(* PLC project Plc Structured Text Cheatsheet, CODESYS CODESYS V3.5 SP16, author Toni Kucic *)
(* stored: creationDateTime 2022-05-27T13:55:14.4433933, version 1.0, modificationDateTime 2022-05-27T13:55:00.8059953, organization TK Automation *)
(* Cheatsheet for programming a PLC in IEC61131-3 Structured text. Contains usage of operators and common functions. *)

TYPE dtTestStruct : STRUCT
  dummy1 : USINT := 255;
  Elem1 : INT := -1;
  Id : DWORD := 215215126;
  IdText : STRING := 'Testing for speed';
  dummy2 : ARRAY[0..11] OF DWORD;
  dummy4 : BOOL := FALSE;
  dummy5 : STRING(255) := 'Big array';
  dummy6 : LINT := 1211212723838939;
END_STRUCT;
END_TYPE

PROGRAM floatingPointOperations
  VAR CONSTANT
    cNrRuns : USINT := 5;
    cRepeatCalcTimes : UDINT := 10000000;  (* 10 Million times *)
  END_VAR
  VAR
    vResultsA : ARRAY[0..cNrRuns] OF LTIME;  (* Boiler plate variables for test *)
    vResultsB : ARRAY[0..cNrRuns] OF LTIME;
    vResultsC : ARRAY[0..cNrRuns] OF LTIME;
    vResultsD : ARRAY[0..cNrRuns] OF LTIME;
    vResultsE : ARRAY[0..cNrRuns] OF LTIME;
    vResultsF : ARRAY[0..cNrRuns] OF LTIME;
    vResultsG : ARRAY[0..cNrRuns] OF LTIME;
    vResultsH : ARRAY[0..cNrRuns] OF LTIME;
    vResultsI : ARRAY[0..cNrRuns] OF LTIME;
    vResultsAAVG : LTIME;
    vResultsBAVG : LTIME;
    vResultsCAVG : LTIME;
    vResultsDAVG : LTIME;
    vResultsEAVG : LTIME;
    vResultsFAVG : LTIME;
    vResultsGAVG : LTIME;
    vResultsHAVG : LTIME;
    vResultsIAVG : LTIME;
    vWayAOldTime : LTIME;
    vWayBOldTime : LTIME;
    vWayCOldTime : LTIME;
    vWayDOldTime : LTIME;
    vWayEOldTime : LTIME;
    vWayFOldTime : LTIME;
    vWayGOldTime : LTIME;
    vWayHOldTime : LTIME;
    vWayIOldTime : LTIME;
    vWayAExecTime : LTIME;
    vWayBExecTime : LTIME;
    vWayCExecTime : LTIME;
    vWayDExecTime : LTIME;
    vWayEExecTime : LTIME;
    vWayFExecTime : LTIME;
    vWayGExecTime : LTIME;
    vWayHExecTime : LTIME;
    vWayIExecTime : LTIME;
    i : UDINT;
    vRunsCompleted : USINT := 0;
    vInteger1 : INT := 1234;  (* Test vars *)
    vInteger2 : INT := 4231;
    vReal1 : REAL := 1234.4231;
    vReal2 : REAL := 4231.1234;
    vInteger3 : DINT := 1234;
    vInteger4 : DINT := 4231;
    vResult1 : INT;
    vResult2 : REAL;
    vResult3 : DINT;
    vResult4 : INT;
    vResult5 : REAL;
    vResult6 : DINT;
    vResult7 : INT;
    vResult8 : REAL;
    vResult9 : DINT;
  END_VAR

            IF vRunsCompleted > cNrRuns THEN
	vResultsAAVG := calcAvg(vResultsA); //Time to add two integers 10 milion times
	vResultsBAVG := calcAvg(vResultsB); //Time to add two reals 10 milion times
	vResultsCAVG := calcAvg(vResultsC); //Time to add two DINTs (32b INT) 10 milion times
	vResultsDAVG := calcAvg(vResultsD); //Time to multiply two integers 10 milion times
	vResultsEAVG := calcAvg(vResultsE); //Time to multiply two reals 10 milion times
	vResultsFAVG := calcAvg(vResultsF); //Time to multiply two DINTs (32b INT) 10 milion times
	vResultsGAVG := calcAvg(vResultsG); //Time to divide two integers 10 milion times
	vResultsHAVG := calcAvg(vResultsH); //Time to divide two reals 10 milion times
	vResultsIAVG := calcAvg(vResultsI); //Time to divide two DINTs (32b INT) 10 milion times
	RETURN;
END_IF

//------------CALCULATION A -------------------
vWayAOldTime := LTIME();
FOR i:= 0 TO cRepeatCalcTimes DO
	vResult1 := vInteger1 + vInteger2;
END_FOR
vWayAExecTime := LTIME() - vWayAOldTime;

//------------CALCULATION B -------------------
vWayBOldTime := LTIME();
FOR i:= 0 TO cRepeatCalcTimes DO
	vResult2 := vReal1 + vReal2;
END_FOR
vWayBExecTime := LTIME() - vWayBOldTime;

//------------CALCULATION C -------------------
vWayCOldTime := LTIME();
FOR i:= 0 TO cRepeatCalcTimes DO
	vResult3 := vInteger3 + vInteger4;
END_FOR
vWayCExecTime := LTIME() - vWayCOldTime;

//------------CALCULATION D -------------------
vWayDOldTime := LTIME();
FOR i:= 0 TO cRepeatCalcTimes DO
	vResult4 := vInteger1 * vInteger2;
END_FOR
vWayDExecTime := LTIME() - vWayDOldTime;

//------------CALCULATION E -------------------
vWayEOldTime := LTIME();
FOR i:= 0 TO cRepeatCalcTimes DO
	vResult5 := vReal1 * vReal2;
END_FOR
vWayEExecTime := LTIME() - vWayEOldTime;

//------------CALCULATION F -------------------
vWayFOldTime := LTIME();
FOR i:= 0 TO cRepeatCalcTimes DO
	vResult6 := vInteger3 * vInteger4;
END_FOR
vWayFExecTime := LTIME() - vWayFOldTime;

//------------CALCULATION G -------------------
vWayGOldTime := LTIME();
FOR i:= 0 TO cRepeatCalcTimes DO
	vResult7 := vInteger1 / vInteger2;
END_FOR
vWayGExecTime := LTIME() - vWayGOldTime;

//------------CALCULATION H -------------------
vWayHOldTime := LTIME();
FOR i:= 0 TO cRepeatCalcTimes DO
	vResult8 := vReal1 / vReal2;
END_FOR
vWayHExecTime := LTIME() - vWayHOldTime;

//------------CALCULATION I -------------------
vWayIOldTime := LTIME();
FOR i:= 0 TO cRepeatCalcTimes DO
	vResult9 := vInteger3 / vInteger4;
END_FOR
vWayIExecTime := LTIME() - vWayIOldTime;


//------------CATCH RESULTS---------------------
vResultsA[vRunsCompleted] := vWayAExecTime;
vResultsB[vRunsCompleted] := vWayBExecTime;
vResultsC[vRunsCompleted] := vWayCExecTime;
vResultsD[vRunsCompleted] := vWayDExecTime;
vResultsE[vRunsCompleted] := vWayEExecTime;
vResultsF[vRunsCompleted] := vWayFExecTime;
vResultsG[vRunsCompleted] := vWayGExecTime;
vResultsH[vRunsCompleted] := vWayHExecTime;
vResultsI[vRunsCompleted] := vWayIExecTime;
vRunsCompleted := vRunsCompleted + 1;

          
END_PROGRAM

FUNCTION addTwoInts : INT
  VAR_IN_OUT
    int1 : INT;
    int2 : INT;
  END_VAR

            addTwoInts := int1 + int2;
          
END_FUNCTION

PROGRAM FunctionOverhead
  VAR CONSTANT
    cNrRuns : USINT := 4;
    cRepeatCalcTimes : UDINT := 10000000;  (* Million times *)
  END_VAR
  VAR
    vResultsA : ARRAY[0..cNrRuns] OF LTIME;  (* Boiler plate variables for test *)
    vResultsB : ARRAY[0..cNrRuns] OF LTIME;
    vResultsC : ARRAY[0..cNrRuns] OF LTIME;
    vResultsAAVG : LTIME;
    vResultsBAVG : LTIME;
    vResultsCAVG : LTIME;
    vWayAOldTime : LTIME;
    vWayBOldTime : LTIME;
    vWayCOldTime : LTIME;
    vWayAExecTime : LTIME;
    vWayBExecTime : LTIME;
    vWayCExecTime : LTIME;
    i : UDINT;
    vRunsCompleted : USINT := 0;
    vInt1 : INT := 1;  (* Test vars *)
    vInt2 : INT := 2;
    vResult1 : INT;
    vResult2 : INT;
    vResult3 : INT;
  END_VAR

            IF vRunsCompleted > cNrRuns THEN
	vResultsAAVG := calcAvg(vResultsA); //Operands
	vResultsBAVG := calcAvg(vResultsB); //User function
	vResultsCAVG := calcAvg(vResultsC); //PRG method
	RETURN;
END_IF
	
//------------CALCULATION A -------------------
vWayAOldTime := LTIME();
FOR i:= 0 TO cRepeatCalcTimes DO
	vResult1 := vInt1 + vInt2;
END_FOR
vWayAExecTime := LTIME() - vWayAOldTime;

//------------CALCULATION B -------------------
vWayBOldTime := LTIME();
FOR i:= 0 TO cRepeatCalcTimes DO
	vResult2 := addTwoInts(vInt1, vInt2);
END_FOR
vWayBExecTime := LTIME() - vWayBOldTime;

//------------CALCULATION C -------------------
vWayCOldTime := LTIME();
FOR i:= 0 TO cRepeatCalcTimes DO
	vResult3 := addTwoNumbers(vInt1, vInt2);
END_FOR
vWayCExecTime := LTIME() - vWayCOldTime;

//------------CATCH RESULTS---------------------
vResultsA[vRunsCompleted] := vWayAExecTime;
vResultsB[vRunsCompleted] := vWayBExecTime;
vResultsC[vRunsCompleted] := vWayCExecTime;
vRunsCompleted := vRunsCompleted + 1;

          

METHOD addTwoNumbers : INT
  VAR_INPUT
    int1 : INT;
    int2 : INT;
  END_VAR
                  addTwoNumbers := int1 + int2;
                
END_METHOD
END_PROGRAM

PROGRAM ImpactOfDynamicArrays
  VAR CONSTANT
    cNrRuns : USINT := 4;
    cRepeatCalcTimes : UDINT := 1000000;  (* Million times *)
  END_VAR
  VAR
    vResultsA : ARRAY[0..cNrRuns] OF LTIME;  (* Boiler plate variables for test *)
    vResultsB : ARRAY[0..cNrRuns] OF LTIME;
    vResultsAAVG : LTIME;
    vResultsBAVG : LTIME;
    vWayAOldTime : LTIME;
    vWayAExecTime : LTIME;
    vWayBOldTime : LTIME;
    vWayBExecTime : LTIME;
    i : UDINT;
    vRunsCompleted : USINT := 0;
    vAvgTimeFun : LTIME;  (* Test vars *)
    vAvgTimeHardCoded : LTIME;
    vTimes : ARRAY[0..9] OF LTIME := [LTIME#1ms0us0ns, LTIME#2ms0us0ns, LTIME#3ms0us0ns, LTIME#4ms0us0ns, LTIME#5ms0us0ns, LTIME#6ms0us0ns, LTIME#7ms0us0ns, LTIME#8ms0us0ns, LTIME#9ms0us0ns, LTIME#10ms0us0ns];
    j : USINT;
  END_VAR

            IF vRunsCompleted > cNrRuns THEN
	vResultsAAVG := calcAvg(vResultsA);
	vResultsBAVG := calcAvg(vResultsB);
	RETURN;
END_IF
	
//------------CALCULATION A -------------------
vWayAOldTime := LTIME();
FOR i:= 0 TO cRepeatCalcTimes DO
	vAvgTimeFun := calcAvg(vTimes);
END_FOR
vWayAExecTime := LTIME() - vWayAOldTime;

//------------CALCULATION B -------------------
vWayBOldTime := LTIME();
FOR i:= 0 TO cRepeatCalcTimes DO
	vAvgTimeHardCoded := LTIME#0MS;
	FOR j:= 0 TO 9 DO
		vAvgTimeHardCoded := vAvgTimeHardCoded + vTimes[j];
	END_FOR
	vAvgTimeHardCoded := vAvgTimeHardCoded / j;
END_FOR
vWayBExecTime := LTIME() - vWayBOldTime;

//------------CATCH RESULTS---------------------
vResultsA[vRunsCompleted] := vWayAExecTime;
vResultsB[vRunsCompleted] := vWayBExecTime;
vRunsCompleted := vRunsCompleted + 1;

          
END_PROGRAM

PROGRAM ShlVsMemCpy
  VAR CONSTANT
    cNrRuns : USINT := 4;
    cRepeatCalcTimes : UDINT := 1000000;  (* Million times *)
  END_VAR
  VAR
    vResultsA : ARRAY[0..cNrRuns] OF LTIME;  (* Boiler plate variables for test *)
    vResultsB : ARRAY[0..cNrRuns] OF LTIME;
    vResultsAAVG : LTIME;
    vResultsBAVG : LTIME;
    vWayAOldTime : LTIME;
    vWayAExecTime : LTIME;
    vWayBOldTime : LTIME;
    vWayBExecTime : LTIME;
    i : UDINT;
    vRunsCompleted : USINT := 0;
    vSHRInteger : UINT;  (* Test vars *)
    vMcpyInteger : UINT;
    vBuffer : ARRAY[0..1] OF USINT := [16#55, 16#AA];
    vSHLOldTime : LTIME;
    vMcpyOldTime : LTIME;
    vSHLExecTime : LTIME;
    vMcpyExecTime : LTIME;
  END_VAR

            IF vRunsCompleted > cNrRuns THEN
	vResultsAAVG := calcAvg(vResultsA);
	vResultsBAVG := calcAvg(vResultsB);
	RETURN;
END_IF
	

vWayAOldTime := LTIME();
FOR i:= 0 TO cRepeatCalcTimes DO
	//Assemble an UINT from two USINTs using SHR operator
	vSHRInteger := vBuffer[0] + SHL(vBuffer[1],8);
END_FOR
vWayAExecTime := LTIME() - vWayAOldTime;

vWayBOldTime := LTIME();
FOR i:= 0 TO cRepeatCalcTimes DO
	//Assemble an UINT from two USINTs using MemCpy
	MEMUtils.MemCpy(pbyDest:= ADR(vMcpyInteger), pbySrc:= ADR(vBuffer) , dwSize:= SIZEOF(vMcpyInteger));
END_FOR
vWayBExecTime := LTIME() - vWayBOldTime;

//Results
vResultsA[vRunsCompleted] := vWayAExecTime;
vResultsB[vRunsCompleted] := vWayBExecTime;
vRunsCompleted := vRunsCompleted + 1;

          
END_PROGRAM

FUNCTION calcAVG : LTIME
  VAR_INPUT
    {attribute 'variable_length_array' := 'ARRAY[*] OF LTIME'}
    {attribute 'Dimensions' := '1'}
    Results : POINTER TO LTIME;
  END_VAR
  VAR
    i : DINT;
  END_VAR

            FOR i:= LOWER_BOUND(Results,1) TO UPPER_BOUND(Results,1) DO
	calcAvg := calcAvg + Results[i];
END_FOR
calcAvg := calcAvg / i;
RETURN;
          
END_FUNCTION

PROGRAM MemSetVsDataZeero
  VAR CONSTANT
    cNrRuns : USINT := 4;
    cRepeatCalcTimes : UDINT := 1000000;  (* Million times *)
    cEmptyStruct : dtTestStruct;
  END_VAR
  VAR
    vResultsA : ARRAY[0..cNrRuns] OF LTIME;  (* Boiler plate variables for test *)
    vResultsB : ARRAY[0..cNrRuns] OF LTIME;
    vResultsAAVG : LTIME;
    vResultsBAVG : LTIME;
    vWayAOldTime : LTIME;
    vWayAExecTime : LTIME;
    vWayBOldTime : LTIME;
    vWayBExecTime : LTIME;
    i : UDINT;
    vRunsCompleted : USINT := 0;
    vResultStruct1 : dtTestStruct;  (* Test variables *)
    vResultStruct2 : dtTestStruct;
  END_VAR

            IF vRunsCompleted > cNrRuns THEN
	vResultsAAVG := calcAvg(vResultsA);
	vResultsBAVG := calcAvg(vResultsB);
	RETURN;
END_IF
	
//------------CALCULATION A -------------------
vWayAOldTime := LTIME();
FOR i:= 0 TO cRepeatCalcTimes DO
	//RESET STRUCT WITH A EMPTY STRUCT
	vResultStruct1 := cEmptyStruct;
END_FOR
vWayAExecTime := LTIME() - vWayAOldTime;

//------------CALCULATION B -------------------
vWayBOldTime := LTIME();
FOR i:= 0 TO cRepeatCalcTimes DO
	//RESET STRUCT WITH MEM SET
	MEMUtils.MemSet(pbyBuffer:= ADR(vResultStruct2), byValue:= 16#0 , dwSize:= SIZEOF(vResultStruct2));
END_FOR
vWayBExecTime := LTIME() - vWayBOldTime;

//------------CATCH RESULTS---------------------
vResultsA[vRunsCompleted] := vWayAExecTime;
vResultsB[vRunsCompleted] := vWayBExecTime;
vRunsCompleted := vRunsCompleted + 1;

          
END_PROGRAM

PROGRAM execSpeedOfLanguageTypes
  VAR CONSTANT
    cNrRuns : USINT := 4;
    cRepeatCalcTimes : UDINT := 10000000;  (* Million times *)
  END_VAR
  VAR
    vResultsA : ARRAY[0..cNrRuns] OF LTIME;  (* Boiler plate variables for test *)
    vResultsB : ARRAY[0..cNrRuns] OF LTIME;
    vResultsC : ARRAY[0..cNrRuns] OF LTIME;
    vResultsAAVG : LTIME;
    vResultsBAVG : LTIME;
    vResultsCAVG : LTIME;
    vWayAOldTime : LTIME;
    vWayBOldTime : LTIME;
    vWayCOldTime : LTIME;
    vWayAExecTime : LTIME;
    vWayBExecTime : LTIME;
    vWayCExecTime : LTIME;
    i : UDINT;
    vRunsCompleted : USINT := 0;
    vInt1 : INT := 1;  (* Test vars *)
    vInt2 : INT := 2;
    vResult1 : INT;
    vResult2 : INT;
    vResult3 : INT;
  END_VAR

            IF vRunsCompleted > cNrRuns THEN
	vResultsAAVG := calcAvg(vResultsA); //User function Ladder
	vResultsBAVG := calcAvg(vResultsB); //User function ST
	vResultsCAVG := calcAvg(vResultsC); //User function FBD
	RETURN;
END_IF
	
//------------CALCULATION A -------------------
vWayAOldTime := LTIME();
FOR i:= 0 TO cRepeatCalcTimes DO
	vResult1 := addTwoIntsLadder(vInt1, vInt2);
END_FOR
vWayAExecTime := LTIME() - vWayAOldTime;

//------------CALCULATION B -------------------
vWayBOldTime := LTIME();
FOR i:= 0 TO cRepeatCalcTimes DO
	vResult2 := addTwoIntsST(vInt1, vInt2);
END_FOR
vWayBExecTime := LTIME() - vWayBOldTime;

//------------CALCULATION C -------------------
vWayCOldTime := LTIME();
FOR i:= 0 TO cRepeatCalcTimes DO
	vResult3 := addTwoIntsFBD(vInt1, vInt2);
END_FOR
vWayCExecTime := LTIME() - vWayCOldTime;

//------------CATCH RESULTS---------------------
vResultsA[vRunsCompleted] := vWayAExecTime;
vResultsB[vRunsCompleted] := vWayBExecTime;
vResultsC[vRunsCompleted] := vWayCExecTime;
vRunsCompleted := vRunsCompleted + 1;

          
END_PROGRAM

FUNCTION addTwoIntsLadder : INT
  VAR_INPUT
    Int1 : INT;
    Int2 : INT;
  END_VAR

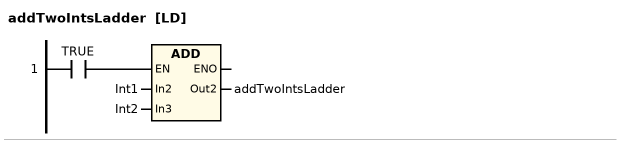
(* LD diagram, written out as Structured Text *)

IF TRUE THEN addTwoIntsLadder := Int1 + Int2; END_IF;
END_FUNCTION

FUNCTION addTwoIntsST : INT
  VAR_INPUT
    int1 : INT;
    int2 : INT;
  END_VAR

            addTwoIntsST := int1 + int2;
          
END_FUNCTION

FUNCTION addTwoIntsFBD : INT
  VAR_INPUT
    int1 : INT;
    int2 : INT;
  END_VAR

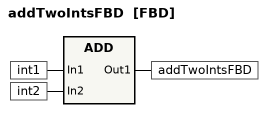
(* FBD diagram, written out as Structured Text *)
addTwoIntsFBD := int1 + int2;
END_FUNCTION

PROGRAM stringOperations
  VAR CONSTANT
    cNrRuns : USINT := 4;
    cRepeatCalcTimes : UDINT := 1000;  (* Million times *)
  END_VAR
  VAR
    vResultsA : ARRAY[0..cNrRuns] OF LTIME;  (* Boiler plate variables for test *)
    vResultsB : ARRAY[0..cNrRuns] OF LTIME;
    vResultsC : ARRAY[0..cNrRuns] OF LTIME;
    vResultsD : ARRAY[0..cNrRuns] OF LTIME;
    vResultsE : ARRAY[0..cNrRuns] OF LTIME;
    vResultsF : ARRAY[0..cNrRuns] OF LTIME;
    vResultsAAVG : LTIME;  (* Time to copy a string[255] 1000 times *)
    vResultsBAVG : LTIME;  (* Time to copy a string 1000 times *)
    vResultsCAVG : LTIME;  (* Time to concatenate 1000 characters with STRING *)
    vResultsDAVG : LTIME;  (* Time to concatenate 1000 characters with STRING[255] *)
    vResultsEAVG : LTIME;  (* Time to copy a BYTE 1000 times *)
    vResultsFAVG : LTIME;  (* Time to copy an array of 255 BYTE 1000 times *)
    vWayAOldTime : LTIME;
    vWayBOldTime : LTIME;
    vWayCOldTime : LTIME;
    vWayDOldTime : LTIME;
    vWayEOldTime : LTIME;
    vWayFOldTime : LTIME;
    vWayAExecTime : LTIME;
    vWayBExecTime : LTIME;
    vWayCExecTime : LTIME;
    vWayDExecTime : LTIME;
    vWayEExecTime : LTIME;
    vWayFExecTime : LTIME;
    i : UDINT;
    vRunsCompleted : USINT := 0;
    vString1 : STRING(255) := 'Test string1';  (* Test vars *)
    vString2 : STRING := 'Test string2';
    vString3 : STRING := 'a';
    vString4 : STRING := 'a';
    vByte : BYTE := 16#FF;
    vArrByte : ARRAY[0..255] OF BYTE;
    vResult1 : STRING(255);
    vResult2 : STRING;
    vResult3 : STRING;
    vResult4 : STRING(255);
    vResult5 : BYTE;
    vResult6 : ARRAY[0..255] OF BYTE;
    vSizes : ARRAY[0..3] OF UDINT;
  END_VAR

            IF vRunsCompleted > cNrRuns THEN
	vResultsAAVG := calcAvg(vResultsA); //Time to copy a string[255] 1000 times
	vResultsBAVG := calcAvg(vResultsB); //Time to copy a string 1000 times
	vResultsCAVG := calcAvg(vResultsC); //Time to concatenate 1000 characters with STRING
	vResultsDAVG := calcAvg(vResultsD); //Time to concatenate 1000  characters with STRING[255]
	vResultsEAVG := calcAvg(vResultsE); //Time to move a byte 1000 times
	vResultsFAVG := calcAvg(vResultsF); //Time to copy an array of 255 BYTE 1000 times
	RETURN;
END_IF

vSizes[0] := SIZEOF(vString1); //Size is 255 characters + zero char
vSizes[1] := SIZEOF(vString2); //Size is 80 characters + zero char, default if no size specified
vSizes[2] := SIZEOF(vResult3); //Size is 81, even though we concatenated 1000 characters. The rest were chopped off
vSizes[3] := SIZEOF(vResult4); //Size is expected 256, other 744 characters chopped off

//------------CALCULATION A -------------------
vWayAOldTime := LTIME();
FOR i:= 0 TO cRepeatCalcTimes DO
	vResult1 := vString1;
END_FOR
vWayAExecTime := LTIME() - vWayAOldTime;

//------------CALCULATION B -------------------
vWayBOldTime := LTIME();
FOR i:= 0 TO cRepeatCalcTimes DO
	vResult2 := vString2;
END_FOR
vWayBExecTime := LTIME() - vWayBOldTime;

//------------CALCULATION C -------------------
vWayCOldTime := LTIME();
FOR i:= 0 TO cRepeatCalcTimes DO
	vResult3 := CONCAT(vResult3, vString3);
END_FOR
vWayCExecTime := LTIME() - vWayCOldTime;

//------------CALCULATION D -------------------
vWayDOldTime := LTIME();
FOR i:= 0 TO cRepeatCalcTimes DO
	vResult4 := CONCAT(vResult4, vString4);
END_FOR
vWayDExecTime := LTIME() - vWayDOldTime;

//------------CALCULATION E -------------------
vWayEOldTime := LTIME();
FOR i:= 0 TO cRepeatCalcTimes DO
	vResult5 := vByte;
END_FOR
vWayEExecTime := LTIME() - vWayEOldTime;

//------------CALCULATION F -------------------
vWayFOldTime := LTIME();
FOR i:= 0 TO cRepeatCalcTimes DO
	vResult6 := vArrByte;
END_FOR
vWayFExecTime := LTIME() - vWayFOldTime;

//------------CATCH RESULTS---------------------
vResultsA[vRunsCompleted] := vWayAExecTime;
vResultsB[vRunsCompleted] := vWayBExecTime;
vResultsC[vRunsCompleted] := vWayCExecTime;
vResultsD[vRunsCompleted] := vWayDExecTime;
vResultsE[vRunsCompleted] := vWayEExecTime;
vResultsF[vRunsCompleted] := vWayFExecTime;
vRunsCompleted := vRunsCompleted + 1;

          
END_PROGRAM

PROGRAM checkingBools
  VAR CONSTANT
    cNrRuns : USINT := 5;
    cRepeatCalcTimes : UDINT := 10000;  (* 10 Million times *)
  END_VAR
  VAR
    vResultsA : ARRAY[0..cNrRuns] OF LTIME;  (* Boiler plate variables for test *)
    vResultsB : ARRAY[0..cNrRuns] OF LTIME;
    vResultsC : ARRAY[0..cNrRuns] OF LTIME;
    vResultsD : ARRAY[0..cNrRuns] OF LTIME;
    vResultsE : ARRAY[0..cNrRuns] OF LTIME;
    vResultsAAVG : LTIME;
    vResultsBAVG : LTIME;
    vResultsCAVG : LTIME;
    vResultsDAVG : LTIME;
    vResultsEAVG : LTIME;
    vWayAOldTime : LTIME;
    vWayBOldTime : LTIME;
    vWayCOldTime : LTIME;
    vWayDOldTime : LTIME;
    vWayEOldTime : LTIME;
    vWayAExecTime : LTIME;
    vWayBExecTime : LTIME;
    vWayCExecTime : LTIME;
    vWayDExecTime : LTIME;
    vWayEExecTime : LTIME;
    i : UDINT;
    vRunsCompleted : USINT := 0;
    vBool : BOOL := TRUE;  (* Test vars *)
    vResult : BOOL;
    vCounter : UINT := 0;
    vCastedUint : UINT;
  END_VAR

            IF vRunsCompleted > cNrRuns THEN
	vResultsAAVG := calcAvg(vResultsA); //Time to run IF vBool = TRUE THEN 1 000 000 times
	vResultsBAVG := calcAvg(vResultsB); //Time to run IF vBool THEN 1 000 000 times
	vResultsCAVG := calcAvg(vResultsC); //Time to increment a counter using if sentence 1 000 000 times
	vResultsDAVG := calcAvg(vResultsD); //Time to increment a counter using bool to UINT 1 000 000 times
	vResultsEAVG := calcAvg(vResultsE); //Time to cast a bool to UINT 1 000 000 times
	RETURN;
END_IF

//------------CALCULATION A -------------------
vWayAOldTime := LTIME();
//FOR i:= 0 TO cRepeatCalcTimes DO
	IF vBool = TRUE THEN
		vResult := vBool;
	END_IF
//END_FOR
vWayAExecTime := LTIME() - vWayAOldTime;

//------------CALCULATION B -------------------
vWayBOldTime := LTIME();
//FOR i:= 0 TO cRepeatCalcTimes DO
	IF vBool THEN
		vResult := vBool;
	END_IF
//END_FOR
vWayBExecTime := LTIME() - vWayBOldTime;

//------------CALCULATION C -------------------
vWayCOldTime := LTIME();
//FOR i:= 0 TO cRepeatCalcTimes DO
	IF vBool THEN
		vCounter := vCounter + 1;
	END_IF
//END_FOR
vWayCExecTime := LTIME() - vWayCOldTime;

//------------CALCULATION D -------------------
vWayDOldTime := LTIME();
//FOR i:= 0 TO cRepeatCalcTimes DO
	vCounter := vCounter + BOOL_TO_UINT(vBool);
//END_FOR
vWayDExecTime := LTIME() - vWayDOldTime;

//------------CALCULATION D -------------------
vWayEOldTime := LTIME();
//FOR i:= 0 TO cRepeatCalcTimes DO
	;vCastedUint := BOOL_TO_UINT(vBool);
//END_FOR
vWayEExecTime := LTIME() - vWayEOldTime;

//------------CATCH RESULTS---------------------
vResultsA[vRunsCompleted] := vWayAExecTime;
vResultsB[vRunsCompleted] := vWayBExecTime;
vResultsC[vRunsCompleted] := vWayCExecTime;
vResultsD[vRunsCompleted] := vWayDExecTime;
vResultsE[vRunsCompleted] := vWayEExecTime;
vRunsCompleted := vRunsCompleted + 1;

          
END_PROGRAM

PROGRAM caseVsIfElsif
  VAR CONSTANT
    cNrRuns : USINT := 5;
    cRepeatCalcTimes : UDINT := 10000000;  (* 10 Million times *)
  END_VAR
  VAR
    vResultsA : ARRAY[0..cNrRuns] OF LTIME;  (* Boiler plate variables for test *)
    vResultsB : ARRAY[0..cNrRuns] OF LTIME;
    vResultsC : ARRAY[0..cNrRuns] OF LTIME;
    vResultsD : ARRAY[0..cNrRuns] OF LTIME;
    vResultsE : ARRAY[0..cNrRuns] OF LTIME;
    vResultsF : ARRAY[0..cNrRuns] OF LTIME;
    vResultsAAVG : LTIME;
    vResultsBAVG : LTIME;
    vResultsCAVG : LTIME;
    vResultsDAVG : LTIME;
    vResultsEAVG : LTIME;
    vResultsFAVG : LTIME;
    vWayAOldTime : LTIME;
    vWayBOldTime : LTIME;
    vWayCOldTime : LTIME;
    vWayDOldTime : LTIME;
    vWayEOldTime : LTIME;
    vWayFOldTime : LTIME;
    vWayAExecTime : LTIME;
    vWayBExecTime : LTIME;
    vWayCExecTime : LTIME;
    vWayDExecTime : LTIME;
    vWayEExecTime : LTIME;
    vWayFExecTime : LTIME;
    i : UDINT;
    vRunsCompleted : USINT := 0;
    vFirstIndex : INT := 15;  (* Test vars *)
    vMiddleIndex : INT := 50;
    vLastIndex : INT := 99;
    vResultFirst : INT;  (* Should be 0 *)
    vResultMiddle : INT;  (* Should be 50 *)
    vResultLast : INT;  (* Should be 99 *)
  END_VAR

            IF vRunsCompleted > cNrRuns THEN
	vResultsAAVG := calcAvg(vResultsA); //Time to run first branch of IF ELSIF 1 000 000 times
	vResultsBAVG := calcAvg(vResultsB); //Time to run middle branch of IF ELSIF 1 000 000 times
	vResultsCAVG := calcAvg(vResultsC); //Time to run last branch of IF ELSIF 1 000 000 times
	vResultsDAVG := calcAvg(vResultsD); //Time to run first branch of CASE 1 000 000 times
	vResultsEAVG := calcAvg(vResultsE); //Time to run middle branch of CASE 1 000 000 times
	vResultsFAVG := calcAvg(vResultsF); //Time to run last branch of CASE 1 000 000 times
	RETURN;
END_IF

//------------CALCULATION A -------------------
vWayAOldTime := LTIME();
FOR i:= 0 TO cRepeatCalcTimes DO
	vResultFirst := returnIndexIfElsif(vFirstIndex);
END_FOR
vWayAExecTime := LTIME() - vWayAOldTime;

//------------CALCULATION B -------------------
vWayBOldTime := LTIME();
FOR i:= 0 TO cRepeatCalcTimes DO
	vResultMiddle := returnIndexIfElsif(vMiddleIndex);
END_FOR
vWayBExecTime := LTIME() - vWayBOldTime;

//------------CALCULATION C -------------------
vWayCOldTime := LTIME();
FOR i:= 0 TO cRepeatCalcTimes DO
	vResultLast := returnIndexIfElsif(vLastIndex);
END_FOR
vWayCExecTime := LTIME() - vWayCOldTime;

//------------CALCULATION D -------------------
vWayDOldTime := LTIME();
FOR i:= 0 TO cRepeatCalcTimes DO
	vResultFirst := returnIndexCase(vFirstIndex);
END_FOR
vWayDExecTime := LTIME() - vWayDOldTime;

//------------CALCULATION E -------------------
vWayEOldTime := LTIME();
FOR i:= 0 TO cRepeatCalcTimes DO
	vResultMiddle := returnIndexCase(vMiddleIndex);
END_FOR
vWayEExecTime := LTIME() - vWayEOldTime;

//------------CALCULATION F -------------------
vWayFOldTime := LTIME();
FOR i:= 0 TO cRepeatCalcTimes DO
	vResultLast := returnIndexCase(vLastIndex);
END_FOR
vWayFExecTime := LTIME() - vWayFOldTime;

//------------CATCH RESULTS---------------------
vResultsA[vRunsCompleted] := vWayAExecTime;
vResultsB[vRunsCompleted] := vWayBExecTime;
vResultsC[vRunsCompleted] := vWayCExecTime;
vResultsD[vRunsCompleted] := vWayDExecTime;
vResultsE[vRunsCompleted] := vWayEExecTime;
vResultsF[vRunsCompleted] := vWayFExecTime;

vRunsCompleted := vRunsCompleted + 1;

          

METHOD returnIndexIfElsif : INT
  VAR_INPUT
    searchValue : INT;
  END_VAR
                  IF searchValue = 0 THEN
        returnIndexIfElsif:=0;
        RETURN;

ELSIF searchValue = 1 THEN
        returnIndexIfElsif:= 1;
        RETURN;

ELSIF searchValue = 2 THEN
        returnIndexIfElsif:= 2;
        RETURN;

ELSIF searchValue = 3 THEN
        returnIndexIfElsif:= 3;
        RETURN;

ELSIF searchValue = 4 THEN
        returnIndexIfElsif:= 4;
        RETURN;

ELSIF searchValue = 5 THEN
        returnIndexIfElsif:= 5;
        RETURN;

ELSIF searchValue = 6 THEN
        returnIndexIfElsif:= 6;
        RETURN;

ELSIF searchValue = 7 THEN
        returnIndexIfElsif:= 7;
        RETURN;

ELSIF searchValue = 8 THEN
        returnIndexIfElsif:= 8;
        RETURN;

ELSIF searchValue = 9 THEN
        returnIndexIfElsif:= 9;
        RETURN;

ELSIF searchValue = 10 THEN
        returnIndexIfElsif:= 10;
        RETURN;

ELSIF searchValue = 11 THEN
        returnIndexIfElsif:= 11;
        RETURN;

ELSIF searchValue = 12 THEN
        returnIndexIfElsif:= 12;
        RETURN;

ELSIF searchValue = 13 THEN
        returnIndexIfElsif:= 13;
        RETURN;

ELSIF searchValue = 14 THEN
        returnIndexIfElsif:= 14;
        RETURN;

ELSIF searchValue = 15 THEN
        returnIndexIfElsif:= 15;
        RETURN;

ELSIF searchValue = 16 THEN
        returnIndexIfElsif:= 16;
        RETURN;

ELSIF searchValue = 17 THEN
        returnIndexIfElsif:= 17;
        RETURN;

ELSIF searchValue = 18 THEN
        returnIndexIfElsif:= 18;
        RETURN;

ELSIF searchValue = 19 THEN
        returnIndexIfElsif:= 19;
        RETURN;

ELSIF searchValue = 20 THEN
        returnIndexIfElsif:= 20;
        RETURN;

ELSIF searchValue = 21 THEN
        returnIndexIfElsif:= 21;
        RETURN;

ELSIF searchValue = 22 THEN
        returnIndexIfElsif:= 22;
        RETURN;

ELSIF searchValue = 23 THEN
        returnIndexIfElsif:= 23;
        RETURN;

ELSIF searchValue = 24 THEN
        returnIndexIfElsif:= 24;
        RETURN;

ELSIF searchValue = 25 THEN
        returnIndexIfElsif:= 25;
        RETURN;

ELSIF searchValue = 26 THEN
        returnIndexIfElsif:= 26;
        RETURN;

ELSIF searchValue = 27 THEN
        returnIndexIfElsif:= 27;
        RETURN;

ELSIF searchValue = 28 THEN
        returnIndexIfElsif:= 28;
        RETURN;

ELSIF searchValue = 29 THEN
        returnIndexIfElsif:= 29;
        RETURN;

ELSIF searchValue = 30 THEN
        returnIndexIfElsif:= 30;
        RETURN;

ELSIF searchValue = 31 THEN
        returnIndexIfElsif:= 31;
        RETURN;

ELSIF searchValue = 32 THEN
        returnIndexIfElsif:= 32;
        RETURN;

ELSIF searchValue = 33 THEN
        returnIndexIfElsif:= 33;
        RETURN;

ELSIF searchValue = 34 THEN
        returnIndexIfElsif:= 34;
        RETURN;

ELSIF searchValue = 35 THEN
        returnIndexIfElsif:= 35;
        RETURN;

ELSIF searchValue = 36 THEN
        returnIndexIfElsif:= 36;
        RETURN;

ELSIF searchValue = 37 THEN
        returnIndexIfElsif:= 37;
        RETURN;

ELSIF searchValue = 38 THEN
        returnIndexIfElsif:= 38;
        RETURN;

ELSIF searchValue = 39 THEN
        returnIndexIfElsif:= 39;
        RETURN;

ELSIF searchValue = 40 THEN
        returnIndexIfElsif:= 40;
        RETURN;

ELSIF searchValue = 41 THEN
        returnIndexIfElsif:= 41;
        RETURN;

ELSIF searchValue = 42 THEN
        returnIndexIfElsif:= 42;
        RETURN;

ELSIF searchValue = 43 THEN
        returnIndexIfElsif:= 43;
        RETURN;

ELSIF searchValue = 44 THEN
        returnIndexIfElsif:= 44;
        RETURN;

ELSIF searchValue = 45 THEN
        returnIndexIfElsif:= 45;
        RETURN;

ELSIF searchValue = 46 THEN
        returnIndexIfElsif:= 46;
        RETURN;

ELSIF searchValue = 47 THEN
        returnIndexIfElsif:= 47;
        RETURN;

ELSIF searchValue = 48 THEN
        returnIndexIfElsif:= 48;
        RETURN;

ELSIF searchValue = 49 THEN
        returnIndexIfElsif:= 49;
        RETURN;

ELSIF searchValue = 50 THEN
        returnIndexIfElsif:= 50;
        RETURN;

ELSIF searchValue = 51 THEN
        returnIndexIfElsif:= 51;
        RETURN;

ELSIF searchValue = 52 THEN
        returnIndexIfElsif:= 52;
        RETURN;

ELSIF searchValue = 53 THEN
        returnIndexIfElsif:= 53;
        RETURN;

ELSIF searchValue = 54 THEN
        returnIndexIfElsif:= 54;
        RETURN;

ELSIF searchValue = 55 THEN
        returnIndexIfElsif:= 55;
        RETURN;

ELSIF searchValue = 56 THEN
        returnIndexIfElsif:= 56;
        RETURN;

ELSIF searchValue = 57 THEN
        returnIndexIfElsif:= 57;
        RETURN;

ELSIF searchValue = 58 THEN
        returnIndexIfElsif:= 58;
        RETURN;

ELSIF searchValue = 59 THEN
        returnIndexIfElsif:= 59;
        RETURN;

ELSIF searchValue = 60 THEN
        returnIndexIfElsif:= 60;
        RETURN;

ELSIF searchValue = 61 THEN
        returnIndexIfElsif:= 61;
        RETURN;

ELSIF searchValue = 62 THEN
        returnIndexIfElsif:= 62;
        RETURN;

ELSIF searchValue = 63 THEN
        returnIndexIfElsif:= 63;
        RETURN;

ELSIF searchValue = 64 THEN
        returnIndexIfElsif:= 64;
        RETURN;

ELSIF searchValue = 65 THEN
        returnIndexIfElsif:= 65;
        RETURN;

ELSIF searchValue = 66 THEN
        returnIndexIfElsif:= 66;
        RETURN;

ELSIF searchValue = 67 THEN
        returnIndexIfElsif:= 67;
        RETURN;

ELSIF searchValue = 68 THEN
        returnIndexIfElsif:= 68;
        RETURN;

ELSIF searchValue = 69 THEN
        returnIndexIfElsif:= 69;
        RETURN;

ELSIF searchValue = 70 THEN
        returnIndexIfElsif:= 70;
        RETURN;

ELSIF searchValue = 71 THEN
        returnIndexIfElsif:= 71;
        RETURN;

ELSIF searchValue = 72 THEN
        returnIndexIfElsif:= 72;
        RETURN;

ELSIF searchValue = 73 THEN
        returnIndexIfElsif:= 73;
        RETURN;

ELSIF searchValue = 74 THEN
        returnIndexIfElsif:= 74;
        RETURN;

ELSIF searchValue = 75 THEN
        returnIndexIfElsif:= 75;
        RETURN;

ELSIF searchValue = 76 THEN
        returnIndexIfElsif:= 76;
        RETURN;

ELSIF searchValue = 77 THEN
        returnIndexIfElsif:= 77;
        RETURN;

ELSIF searchValue = 78 THEN
        returnIndexIfElsif:= 78;
        RETURN;

ELSIF searchValue = 79 THEN
        returnIndexIfElsif:= 79;
        RETURN;

ELSIF searchValue = 80 THEN
        returnIndexIfElsif:= 80;
        RETURN;

ELSIF searchValue = 81 THEN
        returnIndexIfElsif:= 81;
        RETURN;

ELSIF searchValue = 82 THEN
        returnIndexIfElsif:= 82;
        RETURN;

ELSIF searchValue = 83 THEN
        returnIndexIfElsif:= 83;
        RETURN;

ELSIF searchValue = 84 THEN
        returnIndexIfElsif:= 84;
        RETURN;

ELSIF searchValue = 85 THEN
        returnIndexIfElsif:= 85;
        RETURN;

ELSIF searchValue = 86 THEN
        returnIndexIfElsif:= 86;
        RETURN;

ELSIF searchValue = 87 THEN
        returnIndexIfElsif:= 87;
        RETURN;

ELSIF searchValue = 88 THEN
        returnIndexIfElsif:= 88;
        RETURN;

ELSIF searchValue = 89 THEN
        returnIndexIfElsif:= 89;
        RETURN;

ELSIF searchValue = 90 THEN
        returnIndexIfElsif:= 90;
        RETURN;

ELSIF searchValue = 91 THEN
        returnIndexIfElsif:= 91;
        RETURN;

ELSIF searchValue = 92 THEN
        returnIndexIfElsif:= 92;
        RETURN;

ELSIF searchValue = 93 THEN
        returnIndexIfElsif:= 93;
        RETURN;

ELSIF searchValue = 94 THEN
        returnIndexIfElsif:= 94;
        RETURN;

ELSIF searchValue = 95 THEN
        returnIndexIfElsif:= 95;
        RETURN;

ELSIF searchValue = 96 THEN
        returnIndexIfElsif:= 96;
        RETURN;

ELSIF searchValue = 97 THEN
        returnIndexIfElsif:= 97;
        RETURN;

ELSIF searchValue = 98 THEN
        returnIndexIfElsif:= 98;
        RETURN;

ELSIF searchValue = 99 THEN
        returnIndexIfElsif:= 99;
        RETURN;

END_IF
                
END_METHOD

METHOD returnIndexCase : INT
  VAR_INPUT
    searchValue : INT;
  END_VAR
                  CASE searchValue OF

        0: returnIndexCase := 0;
        RETURN;

        1: returnIndexCase := 1;
        RETURN;

        2: returnIndexCase := 2;
        RETURN;

        3: returnIndexCase := 3;
        RETURN;

        4: returnIndexCase := 4;
        RETURN;

        5: returnIndexCase := 5;
        RETURN;

        6: returnIndexCase := 6;
        RETURN;

        7: returnIndexCase := 7;
        RETURN;

        8: returnIndexCase := 8;
        RETURN;

        9: returnIndexCase := 9;
        RETURN;

        10: returnIndexCase := 10;
        RETURN;

        11: returnIndexCase := 11;
        RETURN;

        12: returnIndexCase := 12;
        RETURN;

        13: returnIndexCase := 13;
        RETURN;

        14: returnIndexCase := 14;
        RETURN;

        15: returnIndexCase := 15;
        RETURN;

        16: returnIndexCase := 16;
        RETURN;

        17: returnIndexCase := 17;
        RETURN;

        18: returnIndexCase := 18;
        RETURN;

        19: returnIndexCase := 19;
        RETURN;

        20: returnIndexCase := 20;
        RETURN;

        21: returnIndexCase := 21;
        RETURN;

        22: returnIndexCase := 22;
        RETURN;

        23: returnIndexCase := 23;
        RETURN;

        24: returnIndexCase := 24;
        RETURN;

        25: returnIndexCase := 25;
        RETURN;

        26: returnIndexCase := 26;
        RETURN;

        27: returnIndexCase := 27;
        RETURN;

        28: returnIndexCase := 28;
        RETURN;

        29: returnIndexCase := 29;
        RETURN;

        30: returnIndexCase := 30;
        RETURN;

        31: returnIndexCase := 31;
        RETURN;

        32: returnIndexCase := 32;
        RETURN;

        33: returnIndexCase := 33;
        RETURN;

        34: returnIndexCase := 34;
        RETURN;

        35: returnIndexCase := 35;
        RETURN;

        36: returnIndexCase := 36;
        RETURN;

        37: returnIndexCase := 37;
        RETURN;

        38: returnIndexCase := 38;
        RETURN;

        39: returnIndexCase := 39;
        RETURN;

        40: returnIndexCase := 40;
        RETURN;

        41: returnIndexCase := 41;
        RETURN;

        42: returnIndexCase := 42;
        RETURN;

        43: returnIndexCase := 43;
        RETURN;

        44: returnIndexCase := 44;
        RETURN;

        45: returnIndexCase := 45;
        RETURN;

        46: returnIndexCase := 46;
        RETURN;

        47: returnIndexCase := 47;
        RETURN;

        48: returnIndexCase := 48;
        RETURN;

        49: returnIndexCase := 49;
        RETURN;

        50: returnIndexCase := 50;
        RETURN;

        51: returnIndexCase := 51;
        RETURN;

        52: returnIndexCase := 52;
        RETURN;

        53: returnIndexCase := 53;
        RETURN;

        54: returnIndexCase := 54;
        RETURN;

        55: returnIndexCase := 55;
        RETURN;

        56: returnIndexCase := 56;
        RETURN;

        57: returnIndexCase := 57;
        RETURN;

        58: returnIndexCase := 58;
        RETURN;

        59: returnIndexCase := 59;
        RETURN;

        60: returnIndexCase := 60;
        RETURN;

        61: returnIndexCase := 61;
        RETURN;

        62: returnIndexCase := 62;
        RETURN;

        63: returnIndexCase := 63;
        RETURN;

        64: returnIndexCase := 64;
        RETURN;

        65: returnIndexCase := 65;
        RETURN;

        66: returnIndexCase := 66;
        RETURN;

        67: returnIndexCase := 67;
        RETURN;

        68: returnIndexCase := 68;
        RETURN;

        69: returnIndexCase := 69;
        RETURN;

        70: returnIndexCase := 70;
        RETURN;

        71: returnIndexCase := 71;
        RETURN;

        72: returnIndexCase := 72;
        RETURN;

        73: returnIndexCase := 73;
        RETURN;

        74: returnIndexCase := 74;
        RETURN;

        75: returnIndexCase := 75;
        RETURN;

        76: returnIndexCase := 76;
        RETURN;

        77: returnIndexCase := 77;
        RETURN;

        78: returnIndexCase := 78;
        RETURN;

        79: returnIndexCase := 79;
        RETURN;

        80: returnIndexCase := 80;
        RETURN;

        81: returnIndexCase := 81;
        RETURN;

        82: returnIndexCase := 82;
        RETURN;

        83: returnIndexCase := 83;
        RETURN;

        84: returnIndexCase := 84;
        RETURN;

        85: returnIndexCase := 85;
        RETURN;

        86: returnIndexCase := 86;
        RETURN;

        87: returnIndexCase := 87;
        RETURN;

        88: returnIndexCase := 88;
        RETURN;

        89: returnIndexCase := 89;
        RETURN;

        90: returnIndexCase := 90;
        RETURN;

        91: returnIndexCase := 91;
        RETURN;

        92: returnIndexCase := 92;
        RETURN;

        93: returnIndexCase := 93;
        RETURN;

        94: returnIndexCase := 94;
        RETURN;

        95: returnIndexCase := 95;
        RETURN;

        96: returnIndexCase := 96;
        RETURN;

        97: returnIndexCase := 97;
        RETURN;

        98: returnIndexCase := 98;
        RETURN;

        99: returnIndexCase := 99;
        RETURN;

END_CASE
                
END_METHOD
END_PROGRAM

CONFIGURATION CODESYS_Control_Win_V3_x64
  RESOURCE Application ON PLC
    TASK Task(INTERVAL := T#100ms, PRIORITY := 1);
    PROGRAM checkingBools WITH Task : checkingBools;
  END_RESOURCE
END_CONFIGURATION
